{attribute 'qualified_only'}
VAR_GLOBAL
		EtherCAT_Master_EJxxxx : EtherCAT_Master_EJxxxx_24234FDA;
		EtherCAT_Master_EKxxxx : EtherCAT_Master_EKxxxx_0AF69055;
END_VAR

(* stored: Version 1.2.0.0, ProductVersion 3.1.4024.9
   GVL GVL_iXlinker: Id {df8692a4-47db-4fbb-92ff-291070518eb9} *)
